{attribute 'TcGenerated'}
// This function has been automatically generated from the project information.
VAR_GLOBAL CONSTANT
    {attribute 'const_non_replaced'}
    {attribute 'linkalways'}
    stLibVersion_lcls_plc_tmo_motion : ST_LibVersion := (iMajor := 1, iMinor := 1, iBuild := 1, iRevision := 0, sVersion := '1.1.1');
END_VAR

(* stored: Version 1.1.0.1, ProductVersion 3.1.4022.18
   GVL Global_Version: Id 32c28e5b-f2fa-4c63-a2d5-d6f1a8e98b40 *)
